FUNCTION_BLOCK FB_ActuatorVelFeedForward
VAR_INPUT
	fActuatorVelocity : LREAL; //Input from inverse velocity kinematics
	fMaxActuatorVelocity : LREAL; //Actuator velocity at full joystick
END_VAR
VAR_OUTPUT
	fVelocityFeedForward : LREAL;
END_VAR
VAR
END_VAR


fVelocityFeedForward := fActuatorVelocity/fMaxActuatorVelocity;

END_FUNCTION_BLOCK

(* stored: Version 1.1.0.1, ProductVersion 3.1.4024.12
   POU FB_ActuatorVelFeedForward: Id {13d3eedd-83ab-46d3-bf50-6c6566c35bda}, SpecialFunc None *)
